// TIA Portal V16 export
// export: Created 2021-04-13T11:10:15.2470049Z, ExportSetting WithDefaults, DisplayName Totally Integrated Automation Portal, DisplayVersion V16, DisplayName TIA Portal Version Control Interface, DisplayVersion V16, DisplayName TIA Portal Openness, DisplayVersion V16, DisplayName STEP 7 Professional, DisplayVersion V16, DisplayName STEP 7 Safety, DisplayVersion V16, DisplayName WinCC Unified SCADA Engineering System, DisplayVersion V16
FUNCTION_BLOCK "setWeightBunker_AM"   // FB3, LAD
{ S7_Optimized_Access := 'TRUE' }
VERSION : 0.1
// Блок уставок, работы упаковочных машин.
// Определяет уставки для бункеров. Дают разрешение на работу бункера.
// Даже если сброшено меньше 
// Говорит о готовности упаковочных машин принять дозу и в какую машину скидывать
// stored: AutoNumber true, IsIECCheckEnabled false, IsRetainMemResEnabled false, MemoryReserve 100, SetENOAutomatically false, UDAEnableTagReadback false
   VAR_INPUT
      enableWork : Bool;   // разрешение работы блока
      weightPack : Real;   // заданный вес упаковки
      measurementError : Real;   // погрешность
      maxWeightBunker : Real;   // максимальный вес в бункере
      mediumWeightProduct : Real;   // средний вес продукта
   END_VAR
   VAR_IN_OUT
      taskWeightBunker : Real;   // целевой вес который ищем в сортировке
      setWeightBunker : Array[0..12] of Real;   // уставки задаваемые в бункера
      isWorkWithBunker : Array[0..12] of Bool;   // разрешение работать с конкретными бункерами
      readyToDrop : Array[0..12] of Bool;   // массив который будет сбрасываться
      YP_ReadyToDrop : Array[0..2] of Bool;   // сигнал говорит о том что в УМ можно 100% чтото скинуть
      stableWeightBunker : Array[0..12] of Real;   // стабильный вес в бункерах
      blockSort : Bool;   // запрещение работы сортировки в блоке сортировки
   END_VAR
   VAR
      measureErrorGramm : Real;   // погрешность измерения в граммах
      dropWeight : Real;   // уже сброшенный вес
      hmiDropWeight : Real;   // отображаемый сброшенный вес на панеле
      hmiMeasurementError : Real;   // отображаемая сброшенная погрешность на панеле
      indexLastDropYP : SInt;   // индекс машины в которую последний раз сбрасывали
      full1 : Array[0..12] of Bool;
      full0 : Array[0..12] of Bool;
      Sort_Real_FB : "Sort_Real";
   END_VAR
   VAR_TEMP
      i : DInt;
      j : DInt;
      k : DInt;
      l : DInt;
      "m" : DInt;
      expX : Real;
      expY : Real;
      tmpNeedWeight : Real;
      tmpc1 : Real;
      tmpc2 : DInt;
      tmpc3 : Real;
      minSearch : Real;   // минимальное найденое число остаточном массиве
      indexMinSearch : DInt;   // индекс минимального числа
      isSearchSuccess : Bool;   // поиск прошел успешно
      indexSearchSuccess : DInt;   // индекс оставшегося идеального кармана
      valueDropBunker : DInt;
      tmpArrNotDrop : Array[0..12] of Real;
      tmpArrWeightNoDrop : Array[0..12] of Real;
      noDrop : Int;
      tmpSumFind : Real;
      indexTmpSumFind : DInt;
   END_VAR
   // full1[1..12] := true;
BEGIN

REGION Network 1 (SCL): переведем погрешность в граммы
   #measureErrorGramm := #measurementError * #weightPack / 100;
END_REGION

REGION Network 2 (SCL): Определяем уставки в карманы и выставляем разрешения работы
   // на основе веса который мы уже сбросили и который будем сбрасывать 
   // а также учитывая веса в рецепте определяем уставки в карманах, целевую уставку для поиска, а также 
   // выставляем разрешения работы по конкретным бункерам
   IF #enableWork THEN

       //*********************************************
       //определение сброшенного веса на основе массивов со стабильными весами
       //и массива ячеек которые должны быть сброшены. Обнуление сброшенного веса в случае 
       //выполнения условия
       //также производим этот расчет только при условии что мы сбросим кудато этот вес
       IF #YP_ReadyToDrop[1] OR #YP_ReadyToDrop[2] THEN
           #i := 0;
           FOR #i := 1 TO 12 DO
               #dropWeight := #dropWeight + BOOL_TO_INT(#readyToDrop[#i]) * #stableWeightBunker[#i];
           END_FOR;
           // #hmiDropWeight := #dropWeight;
           // #hmiMeasurementError := (#weightPack - #dropWeight) / #weightPack;
           IF #dropWeight >= #weightPack THEN
               #dropWeight := 0;
           END_IF;
       END_IF;
       //************************************


       //основное распространение весов, когда выкидываем весь вес за раз
       //

       #expX := #weightPack / 10;//#weightPack / 10;
       #expY := #mediumWeightProduct / 3;

       //если #expX<=MAX_WEIGHT_BUNKER то работаем по стандарту,
       //иначе ограничеваем #expX=MAX_WEIGHT_BUNKER
       IF #expX > #maxWeightBunker THEN
           #expX := #maxWeightBunker;
       END_IF;

       IF #dropWeight = 0 THEN
           // #j := 2;
           // WHILE (6 * #expX) < #weightPack + #j * #expY AND #j <> 0 DO
           //     #j := #j - 1;
           // END_WHILE;
           // #expY := (#expY / 2) * #j;//корректировка #expY
           #taskWeightBunker := #weightPack;//вес для поиска по рецепту
           #isWorkWithBunker := #full1;//разрешаем работу всем линиям

           #setWeightBunker[1] := #setWeightBunker[6] :=
           #setWeightBunker[7] := #setWeightBunker[12] := #expX;

           #setWeightBunker[2] := #setWeightBunker[5] :=
           #setWeightBunker[8] := #setWeightBunker[11] := #expX - #expY;

           #setWeightBunker[3] := #setWeightBunker[4] :=
           #setWeightBunker[9] := #setWeightBunker[10] := #expX - 2 * #expY;

       ELSE//если уже сбрасываем

           #valueDropBunker := 0;//определяем сбрасываем ли мы чтото чтобы запретить
           //перерасчет в этом условии
           //просто на первой итерации как только сюда поступает массив readyToDrop
           //мы выставляем требуемые уставки, а потом запрещаем их изменять
           #k := 0;
           FOR #k := 1 TO 12 DO
               #valueDropBunker := #valueDropBunker + BOOL_TO_SINT(#readyToDrop[#k]);
           END_FOR;

           IF #valueDropBunker > 0 THEN
               //следующий просчет актуален только на итерации перед сбросом веса поэтому 
               //после сброса на конвейер эту часть надо блокировать для изменений
               //
               //только еще надо обыгрывать момент когда сбрасываются сразу 12 бункеров

               #tmpNeedWeight := #weightPack - #dropWeight;//вес остатка

               IF #valueDropBunker < 12 THEN //при сбрасывании всех 12 бункеров
                   //будет другой механизм выдачи разрешений

                   IF #tmpNeedWeight <= #expX THEN //если нужно докинуть меньше чем в одном бункере,то
                       //ищем вес совпадающий с остатком и если такой не находим
                       //то берем минимальную ячейку с весом

                       #minSearch := 99999.9;//берется как минимальное тк такое точно не будет в бункере
                       #k := 0;
                       #isSearchSuccess := false;
                       FOR #k := 1 TO 12 DO//ищем бункер идеально подходящий по весу и параллельно ведем
                           //поиск первого минимального числа

                           IF NOT (#readyToDrop[#k]) THEN
                               IF #stableWeightBunker[#k] < #minSearch THEN
                                   //параллельно ищем минимальное число
                                   #minSearch := #stableWeightBunker[#k];
                                   #indexMinSearch := #k;
                               END_IF;

                               IF (#tmpNeedWeight <= #stableWeightBunker[#k]//проверяем оставшиеся карманы на вес
                                   AND #stableWeightBunker[#k] <= #tmpNeedWeight + #measureErrorGramm / 6) THEN
                                   #isSearchSuccess := true;
                                   #indexSearchSuccess := #k;//сохраняем индекс идеального кармана
                                   EXIT;//выходим из FOR
                               END_IF;
                           END_IF;

                       END_FOR;
                       //если идеальный карман так и не найдем 
                       //берем карман с минимальным весом и перемещаем его индекс в #indexSearchSuccess
                       IF NOT (#isSearchSuccess) THEN
                           #indexSearchSuccess := #indexMinSearch;
                       END_IF;

                       #taskWeightBunker := #tmpNeedWeight;//вес для поиска в сортировке
                       #isWorkWithBunker := #full0;//запрещаем работу всем линиям
                       #isWorkWithBunker[#indexSearchSuccess] := true;//включаем только нужную линию
                       #setWeightBunker[#indexSearchSuccess] := #tmpNeedWeight;
                       #blockSort := true;//выставляем блокировку тк надо будет только сбросить

                   ELSE//если докидывать больше чем в одном бункере
                       #k := 0;//выделяем веса которые не сбрасываются
                       FOR #k := 1 TO 12 DO
                           IF NOT (#readyToDrop[#k]) THEN
                               #noDrop := #noDrop + 1;//колво добавленных элементов
                               #tmpArrNotDrop[#k] := #stableWeightBunker[#k];
                           END_IF;
                       END_FOR;
                       //будем использовать #tmpArrWeightNoDrop для поиска искомых бункеров
                       #tmpArrWeightNoDrop := #tmpArrNotDrop;

                       #Sort_Real_FB("array" := #tmpArrNotDrop);
                       //теперь массив #tmpArrNotDrop отсортирован и числа которые 
                       //мы можем использовать начинаются с индекса (12-noDrop+1)
                       #k := 0;
                       #tmpSumFind := 0;//где храним сумму
                       #indexTmpSumFind := 0;//индекс элемента массива на котором надо остановиться
                       FOR #k := (12 - #noDrop + 1) TO 12 DO
                           #tmpSumFind := #tmpSumFind + #tmpArrNotDrop[#k];
                           IF #tmpSumFind >= #tmpNeedWeight//если попадаем идеально
                               AND #tmpSumFind <= #tmpNeedWeight + #measureErrorGramm THEN
                               #indexTmpSumFind := #k;
                               EXIT;//выходим из FOR
                           END_IF;
                           //если превысили сумму
                           IF #tmpSumFind > #tmpNeedWeight + #measureErrorGramm THEN
                               #indexTmpSumFind := #k - 1;
                               EXIT;
                           END_IF;
                           IF #k = 12 THEN
                               #indexTmpSumFind := #k;
                           END_IF;
                       END_FOR;
                       //теперь проверим чтобы #indexTmpSumFind входил в массив с весами
                       //потому что первый же вес может быть больше того что мы исчем
                       IF #tmpArrNotDrop[#indexTmpSumFind] <> 0 THEN
                           #taskWeightBunker := #tmpNeedWeight;//вес для поиска по рецепту
                           #isWorkWithBunker := #full0;//запрещаем работу всем линиям
                           #blockSort := true;//выставляем блокировку тк надо будет только
                           //дождать сигналов готовности к сортировке сбросить

                           //теперь заполняем массив разрешения работ через поиск весов
                           //и параллельно выставляем уставки
                           IF #tmpSumFind >= #tmpNeedWeight//если попадаем идеально
                               AND #tmpSumFind <= #tmpNeedWeight + #measureErrorGramm THEN
                               //если вес сходился 
                               #l := 0;
                               FOR #l := (12 - #noDrop + 1) TO #indexTmpSumFind DO
                                   #m := 0;
                                   FOR #m := 1 TO 12 DO//ищем отсортированные веса и сопоставляем их индексы
                                       //ищем в заранее сохранненом массивве с весам который не сбрасываются
                                       //и имеют правильные индексы
                                       IF #tmpArrWeightNoDrop[#m] = #tmpArrNotDrop[#l] THEN
                                           #isWorkWithBunker[#m] := true;
                                           #setWeightBunker[#m] := #tmpArrWeightNoDrop[#m];
                                           EXIT;//ищем следующий вес
                                       END_IF;
                                   END_FOR;
                               END_FOR;

                           ELSE //сюда поподем если веса с излишкой или недостаточно 
                               //если вес не сходился
                               #l := 0;
                               FOR #l := (12 - #noDrop + 1) TO #indexTmpSumFind DO
                                   #m := 0;
                                   FOR #m := 1 TO 12 DO
                                       IF #tmpArrWeightNoDrop[#m] = #tmpArrNotDrop[#l] THEN
                                           #isWorkWithBunker[#m] := true;
                                           #setWeightBunker[#m] := #tmpNeedWeight / DINT_TO_INT((#indexTmpSumFind - (12 - #noDrop + 1)));
                                           EXIT;//ищем следующий вес
                                       END_IF;
                                   END_FOR;
                               END_FOR;


                           END_IF;
                           ;

                       END_IF;

                   END_IF;
               ELSE //а теперь что делать если сброшены все 12
                   //надо вводить какойто новый сигнал который сказал бы нагружать бункера только после закрытия? или 
                   //все успеется
                   //!!!обратить внимание на это
                   //

                   //расчитываем сколько бункеров необходимо для сбора оставшегося веса
                   //это делаем на основе максимального веса в бункере
                   //
                   #taskWeightBunker := #tmpNeedWeight;//вес для поиска в сортировке
                   #blockSort := true;//выставляем блокировку тк надо будет только скинуть
                   #tmpc2 := ROUND(#tmpNeedWeight / #maxWeightBunker); //число используемых бункеров
                   #i := 0;
                   FOR #i := 1 TO #tmpc2 DO
                       #isWorkWithBunker[#k] := true;
                       #setWeightBunker[#k] := #tmpNeedWeight / DINT_TO_REAL(#tmpc2);
                   END_FOR;
                   ;
               END_IF;
           END_IF;
       END_IF;


   ELSE
       #isWorkWithBunker := #full0;//запрет на работу все бункерам
   END_IF;
END_REGION
END_FUNCTION_BLOCK
